FUNCTION_BLOCK FB_Mediane_Glissante
VAR_INPUT
END_VAR
VAR_OUTPUT
END_VAR
VAR
END_VAR

END_FUNCTION_BLOCK

(* stored: Version 1.1.0.1
   POU FB_Mediane_Glissante: Id {ceba3ef1-c4f2-4d0e-ad6c-96b3f1d8df8f}, SpecialFunc None *)
